// TIA Portal V19 export
DATA_BLOCK "DB_Recipes"   // DB50
{ S7_Optimized_Access := 'TRUE' }
// stored: AutoNumber false, IsOnlyStoredInLoadMemory true, MemoryReserve 100
   VAR RETAIN
      aRecipe : Array[0..256] of "stRecipe";
   END_VAR
BEGIN
   aRecipe[1].RecipeName := 'Test Flate Plate';
   aRecipe[2].RecipeName := 'Test Carbody Shell';
   aRecipe[3].RecipeName := 'RGCC5';
   aRecipe[4..23].RecipeName := '';
   aRecipe[1].RecipeCbsType := 'Flate plate';
   aRecipe[2].RecipeCbsType := 'Carbody shell';
   aRecipe[3].RecipeCbsType := 'RGC';
   aRecipe[4..5].RecipeCbsType := '';
   aRecipe[7..23].RecipeCbsType := '';
   aRecipe[1].RecipeTrajNumber := 100;
   aRecipe[2].RecipeTrajNumber := 101;
   aRecipe[3].RecipeTrajNumber := 11;
   aRecipe[4..8].RecipeTrajNumber := 0;
   aRecipe[10..23].RecipeTrajNumber := 0;
   aRecipe[1..3].RecipeRawMaterial := 1;
   aRecipe[4..8].RecipeRawMaterial := 0;
   aRecipe[10..23].RecipeRawMaterial := 0;
   aRecipe[4].RecipeLayerType[1].RecipeLayerTypeName := '';
   aRecipe[5].RecipeLayerType[1].RecipeLayerTypeName := '';
   aRecipe[6].RecipeLayerType[1].RecipeLayerTypeName := '';
   aRecipe[7].RecipeLayerType[1].RecipeLayerTypeName := '';
   aRecipe[8].RecipeLayerType[1].RecipeLayerTypeName := '';
   aRecipe[9].RecipeLayerType[1].RecipeLayerTypeName := '';
   aRecipe[10].RecipeLayerType[1].RecipeLayerTypeName := '';
   aRecipe[11].RecipeLayerType[1].RecipeLayerTypeName := '';
   aRecipe[12].RecipeLayerType[1].RecipeLayerTypeName := '';
   aRecipe[13].RecipeLayerType[1].RecipeLayerTypeName := '';
   aRecipe[14].RecipeLayerType[1].RecipeLayerTypeName := '';
   aRecipe[15].RecipeLayerType[1].RecipeLayerTypeName := '';
   aRecipe[16].RecipeLayerType[1].RecipeLayerTypeName := '';
   aRecipe[17].RecipeLayerType[1].RecipeLayerTypeName := '';
   aRecipe[18].RecipeLayerType[1].RecipeLayerTypeName := '';
   aRecipe[19].RecipeLayerType[1].RecipeLayerTypeName := '';
   aRecipe[20].RecipeLayerType[1].RecipeLayerTypeName := '';
   aRecipe[21].RecipeLayerType[1].RecipeLayerTypeName := '';
   aRecipe[22].RecipeLayerType[1].RecipeLayerTypeName := '';
   aRecipe[23].RecipeLayerType[1].RecipeLayerTypeName := '';
   aRecipe[1].RecipeLayerType[1].JobTableLeft[0].SetForceZero := 0;
   aRecipe[1].RecipeLayerType[1].JobTableLeft[1..4].SetForceZero := 100;
   aRecipe[1].RecipeLayerType[2].JobTableLeft[0].SetForceZero := 0;
   aRecipe[1].RecipeLayerType[2].JobTableLeft[1].SetForceZero := 100;
   aRecipe[1].RecipeLayerType[2].JobTableLeft[2..3].SetForceZero := 90;
   aRecipe[2].RecipeLayerType[1].JobTableLeft[0].SetForceZero := 0;
   aRecipe[2].RecipeLayerType[1].JobTableLeft[1].SetForceZero := 50;
   aRecipe[2].RecipeLayerType[2].JobTableLeft[0].SetForceZero := 0;
   aRecipe[2].RecipeLayerType[2].JobTableLeft[1].SetForceZero := 100;
   aRecipe[2].RecipeLayerType[2].JobTableLeft[2..3].SetForceZero := 80;
   aRecipe[3].RecipeLayerType[1].JobTableLeft[0].SetForceZero := 0;
   aRecipe[3].RecipeLayerType[1].JobTableLeft[1..2].SetForceZero := 80;
   aRecipe[3].RecipeLayerType[2].JobTableLeft[0].SetForceZero := 0;
   aRecipe[3].RecipeLayerType[2].JobTableLeft[1].SetForceZero := 80;
   aRecipe[4].RecipeLayerType[1].JobTableLeft[0].SetForceZero := 0;
   aRecipe[4].RecipeLayerType[2].JobTableLeft[0].SetForceZero := 0;
   aRecipe[5].RecipeLayerType[1].JobTableLeft[0].SetForceZero := 0;
   aRecipe[5].RecipeLayerType[2].JobTableLeft[0].SetForceZero := 0;
   aRecipe[6].RecipeLayerType[1].JobTableLeft[0].SetForceZero := 0;
   aRecipe[6].RecipeLayerType[1].JobTableLeft[1].SetForceZero := 20;
   aRecipe[6].RecipeLayerType[2].JobTableLeft[0].SetForceZero := 0;
   aRecipe[6].RecipeLayerType[2].JobTableLeft[1].SetForceZero := 20;
   aRecipe[7].RecipeLayerType[1].JobTableLeft[0].SetForceZero := 0;
   aRecipe[7].RecipeLayerType[2].JobTableLeft[0].SetForceZero := 0;
   aRecipe[8].RecipeLayerType[1].JobTableLeft[0].SetForceZero := 0;
   aRecipe[8].RecipeLayerType[2].JobTableLeft[0].SetForceZero := 0;
   aRecipe[9].RecipeLayerType[1].JobTableLeft[0].SetForceZero := 0;
   aRecipe[9].RecipeLayerType[2].JobTableLeft[0].SetForceZero := 0;
   aRecipe[10].RecipeLayerType[1].JobTableLeft[0].SetForceZero := 0;
   aRecipe[10].RecipeLayerType[2].JobTableLeft[0].SetForceZero := 0;
   aRecipe[11].RecipeLayerType[1].JobTableLeft[0].SetForceZero := 0;
   aRecipe[11].RecipeLayerType[2].JobTableLeft[0].SetForceZero := 0;
   aRecipe[12].RecipeLayerType[1].JobTableLeft[0].SetForceZero := 0;
   aRecipe[12].RecipeLayerType[2].JobTableLeft[0].SetForceZero := 0;
   aRecipe[13].RecipeLayerType[1].JobTableLeft[0].SetForceZero := 0;
   aRecipe[13].RecipeLayerType[2].JobTableLeft[0].SetForceZero := 0;
   aRecipe[14].RecipeLayerType[1].JobTableLeft[0].SetForceZero := 0;
   aRecipe[14].RecipeLayerType[2].JobTableLeft[0].SetForceZero := 0;
   aRecipe[15].RecipeLayerType[1].JobTableLeft[0].SetForceZero := 0;
   aRecipe[15].RecipeLayerType[2].JobTableLeft[0].SetForceZero := 0;
   aRecipe[16].RecipeLayerType[1].JobTableLeft[0].SetForceZero := 0;
   aRecipe[16].RecipeLayerType[2].JobTableLeft[0].SetForceZero := 0;
   aRecipe[17].RecipeLayerType[1].JobTableLeft[0].SetForceZero := 0;
   aRecipe[17].RecipeLayerType[2].JobTableLeft[0].SetForceZero := 0;
   aRecipe[18].RecipeLayerType[1].JobTableLeft[0].SetForceZero := 0;
   aRecipe[18].RecipeLayerType[2].JobTableLeft[0].SetForceZero := 0;
   aRecipe[19].RecipeLayerType[1].JobTableLeft[0].SetForceZero := 0;
   aRecipe[19].RecipeLayerType[2].JobTableLeft[0].SetForceZero := 0;
   aRecipe[20].RecipeLayerType[1].JobTableLeft[0].SetForceZero := 0;
   aRecipe[20].RecipeLayerType[2].JobTableLeft[0].SetForceZero := 0;
   aRecipe[21].RecipeLayerType[1].JobTableLeft[0].SetForceZero := 0;
   aRecipe[21].RecipeLayerType[2].JobTableLeft[0].SetForceZero := 0;
   aRecipe[22].RecipeLayerType[1].JobTableLeft[0].SetForceZero := 0;
   aRecipe[22].RecipeLayerType[2].JobTableLeft[0].SetForceZero := 0;
   aRecipe[23].RecipeLayerType[1].JobTableLeft[0].SetForceZero := 0;
   aRecipe[23].RecipeLayerType[2].JobTableLeft[0].SetForceZero := 0;
   aRecipe[1].RecipeLayerType[1].JobTableLeft[0].SetForceTarget := 0;
   aRecipe[1].RecipeLayerType[1].JobTableLeft[1..4].SetForceTarget := 200;
   aRecipe[1].RecipeLayerType[2].JobTableLeft[0].SetForceTarget := 0;
   aRecipe[1].RecipeLayerType[2].JobTableLeft[1].SetForceTarget := 200;
   aRecipe[1].RecipeLayerType[2].JobTableLeft[2].SetForceTarget := 150;
   aRecipe[1].RecipeLayerType[2].JobTableLeft[3].SetForceTarget := 180;
   aRecipe[2].RecipeLayerType[1].JobTableLeft[0].SetForceTarget := 0;
   aRecipe[2].RecipeLayerType[1].JobTableLeft[1].SetForceTarget := 80;
   aRecipe[2].RecipeLayerType[2].JobTableLeft[0].SetForceTarget := 0;
   aRecipe[2].RecipeLayerType[2].JobTableLeft[1].SetForceTarget := 200;
   aRecipe[2].RecipeLayerType[2].JobTableLeft[3].SetForceTarget := 150;
   aRecipe[3].RecipeLayerType[1].JobTableLeft[0].SetForceTarget := 0;
   aRecipe[3].RecipeLayerType[1].JobTableLeft[1..2].SetForceTarget := 120;
   aRecipe[3].RecipeLayerType[2].JobTableLeft[0].SetForceTarget := 0;
   aRecipe[3].RecipeLayerType[2].JobTableLeft[1].SetForceTarget := 120;
   aRecipe[4].RecipeLayerType[1].JobTableLeft[0].SetForceTarget := 0;
   aRecipe[4].RecipeLayerType[2].JobTableLeft[0].SetForceTarget := 0;
   aRecipe[5].RecipeLayerType[1].JobTableLeft[0].SetForceTarget := 0;
   aRecipe[5].RecipeLayerType[2].JobTableLeft[0].SetForceTarget := 0;
   aRecipe[6].RecipeLayerType[1].JobTableLeft[0].SetForceTarget := 0;
   aRecipe[6].RecipeLayerType[1].JobTableLeft[1].SetForceTarget := 120;
   aRecipe[6].RecipeLayerType[2].JobTableLeft[0].SetForceTarget := 0;
   aRecipe[6].RecipeLayerType[2].JobTableLeft[1].SetForceTarget := 120;
   aRecipe[7].RecipeLayerType[1].JobTableLeft[0].SetForceTarget := 0;
   aRecipe[7].RecipeLayerType[2].JobTableLeft[0].SetForceTarget := 0;
   aRecipe[8].RecipeLayerType[1].JobTableLeft[0].SetForceTarget := 0;
   aRecipe[8].RecipeLayerType[2].JobTableLeft[0].SetForceTarget := 0;
   aRecipe[9].RecipeLayerType[1].JobTableLeft[0].SetForceTarget := 0;
   aRecipe[9].RecipeLayerType[2].JobTableLeft[0].SetForceTarget := 0;
   aRecipe[10].RecipeLayerType[1].JobTableLeft[0].SetForceTarget := 0;
   aRecipe[10].RecipeLayerType[2].JobTableLeft[0].SetForceTarget := 0;
   aRecipe[11].RecipeLayerType[1].JobTableLeft[0].SetForceTarget := 0;
   aRecipe[11].RecipeLayerType[2].JobTableLeft[0].SetForceTarget := 0;
   aRecipe[12].RecipeLayerType[1].JobTableLeft[0].SetForceTarget := 0;
   aRecipe[12].RecipeLayerType[2].JobTableLeft[0].SetForceTarget := 0;
   aRecipe[13].RecipeLayerType[1].JobTableLeft[0].SetForceTarget := 0;
   aRecipe[13].RecipeLayerType[2].JobTableLeft[0].SetForceTarget := 0;
   aRecipe[14].RecipeLayerType[1].JobTableLeft[0].SetForceTarget := 0;
   aRecipe[14].RecipeLayerType[2].JobTableLeft[0].SetForceTarget := 0;
   aRecipe[15].RecipeLayerType[1].JobTableLeft[0].SetForceTarget := 0;
   aRecipe[15].RecipeLayerType[2].JobTableLeft[0].SetForceTarget := 0;
   aRecipe[16].RecipeLayerType[1].JobTableLeft[0].SetForceTarget := 0;
   aRecipe[16].RecipeLayerType[2].JobTableLeft[0].SetForceTarget := 0;
   aRecipe[17].RecipeLayerType[1].JobTableLeft[0].SetForceTarget := 0;
   aRecipe[17].RecipeLayerType[2].JobTableLeft[0].SetForceTarget := 0;
   aRecipe[18].RecipeLayerType[1].JobTableLeft[0].SetForceTarget := 0;
   aRecipe[18].RecipeLayerType[2].JobTableLeft[0].SetForceTarget := 0;
   aRecipe[19].RecipeLayerType[1].JobTableLeft[0].SetForceTarget := 0;
   aRecipe[19].RecipeLayerType[2].JobTableLeft[0].SetForceTarget := 0;
   aRecipe[20].RecipeLayerType[1].JobTableLeft[0].SetForceTarget := 0;
   aRecipe[20].RecipeLayerType[2].JobTableLeft[0].SetForceTarget := 0;
   aRecipe[21].RecipeLayerType[1].JobTableLeft[0].SetForceTarget := 0;
   aRecipe[21].RecipeLayerType[2].JobTableLeft[0].SetForceTarget := 0;
   aRecipe[22].RecipeLayerType[1].JobTableLeft[0].SetForceTarget := 0;
   aRecipe[22].RecipeLayerType[2].JobTableLeft[0].SetForceTarget := 0;
   aRecipe[23].RecipeLayerType[1].JobTableLeft[0].SetForceTarget := 0;
   aRecipe[23].RecipeLayerType[2].JobTableLeft[0].SetForceTarget := 0;
   aRecipe[1].RecipeLayerType[1].JobTableLeft[0].SetTimeRamp := 0;
   aRecipe[1].RecipeLayerType[2].JobTableLeft[0].SetTimeRamp := 0;
   aRecipe[2].RecipeLayerType[1].JobTableLeft[0].SetTimeRamp := 0;
   aRecipe[2].RecipeLayerType[2].JobTableLeft[0].SetTimeRamp := 0;
   aRecipe[3].RecipeLayerType[1].JobTableLeft[0].SetTimeRamp := 0;
   aRecipe[3].RecipeLayerType[2].JobTableLeft[0].SetTimeRamp := 0;
   aRecipe[4].RecipeLayerType[1].JobTableLeft[0].SetTimeRamp := 0;
   aRecipe[4].RecipeLayerType[2].JobTableLeft[0].SetTimeRamp := 0;
   aRecipe[5].RecipeLayerType[1].JobTableLeft[0].SetTimeRamp := 0;
   aRecipe[5].RecipeLayerType[2].JobTableLeft[0].SetTimeRamp := 0;
   aRecipe[6].RecipeLayerType[1].JobTableLeft[0].SetTimeRamp := 0;
   aRecipe[6].RecipeLayerType[2].JobTableLeft[0].SetTimeRamp := 0;
   aRecipe[7].RecipeLayerType[1].JobTableLeft[0].SetTimeRamp := 0;
   aRecipe[7].RecipeLayerType[2].JobTableLeft[0].SetTimeRamp := 0;
   aRecipe[8].RecipeLayerType[1].JobTableLeft[0].SetTimeRamp := 0;
   aRecipe[8].RecipeLayerType[2].JobTableLeft[0].SetTimeRamp := 0;
   aRecipe[9].RecipeLayerType[1].JobTableLeft[0].SetTimeRamp := 0;
   aRecipe[9].RecipeLayerType[2].JobTableLeft[0].SetTimeRamp := 0;
   aRecipe[10].RecipeLayerType[1].JobTableLeft[0].SetTimeRamp := 0;
   aRecipe[10].RecipeLayerType[2].JobTableLeft[0].SetTimeRamp := 0;
   aRecipe[11].RecipeLayerType[1].JobTableLeft[0].SetTimeRamp := 0;
   aRecipe[11].RecipeLayerType[2].JobTableLeft[0].SetTimeRamp := 0;
   aRecipe[12].RecipeLayerType[1].JobTableLeft[0].SetTimeRamp := 0;
   aRecipe[12].RecipeLayerType[2].JobTableLeft[0].SetTimeRamp := 0;
   aRecipe[13].RecipeLayerType[1].JobTableLeft[0].SetTimeRamp := 0;
   aRecipe[13].RecipeLayerType[2].JobTableLeft[0].SetTimeRamp := 0;
   aRecipe[14].RecipeLayerType[1].JobTableLeft[0].SetTimeRamp := 0;
   aRecipe[14].RecipeLayerType[2].JobTableLeft[0].SetTimeRamp := 0;
   aRecipe[15].RecipeLayerType[1].JobTableLeft[0].SetTimeRamp := 0;
   aRecipe[15].RecipeLayerType[2].JobTableLeft[0].SetTimeRamp := 0;
   aRecipe[16].RecipeLayerType[1].JobTableLeft[0].SetTimeRamp := 0;
   aRecipe[16].RecipeLayerType[2].JobTableLeft[0].SetTimeRamp := 0;
   aRecipe[17].RecipeLayerType[1].JobTableLeft[0].SetTimeRamp := 0;
   aRecipe[17].RecipeLayerType[2].JobTableLeft[0].SetTimeRamp := 0;
   aRecipe[18].RecipeLayerType[1].JobTableLeft[0].SetTimeRamp := 0;
   aRecipe[18].RecipeLayerType[2].JobTableLeft[0].SetTimeRamp := 0;
   aRecipe[19].RecipeLayerType[1].JobTableLeft[0].SetTimeRamp := 0;
   aRecipe[19].RecipeLayerType[2].JobTableLeft[0].SetTimeRamp := 0;
   aRecipe[20].RecipeLayerType[1].JobTableLeft[0].SetTimeRamp := 0;
   aRecipe[20].RecipeLayerType[2].JobTableLeft[0].SetTimeRamp := 0;
   aRecipe[21].RecipeLayerType[1].JobTableLeft[0].SetTimeRamp := 0;
   aRecipe[21].RecipeLayerType[2].JobTableLeft[0].SetTimeRamp := 0;
   aRecipe[22].RecipeLayerType[1].JobTableLeft[0].SetTimeRamp := 0;
   aRecipe[22].RecipeLayerType[2].JobTableLeft[0].SetTimeRamp := 0;
   aRecipe[23].RecipeLayerType[1].JobTableLeft[0].SetTimeRamp := 0;
   aRecipe[23].RecipeLayerType[2].JobTableLeft[0].SetTimeRamp := 0;
   aRecipe[1].RecipeLayerType[1].JobTableLeft[0].SetSpeed := 0;
   aRecipe[1].RecipeLayerType[1].JobTableLeft[3..4].SetSpeed := 5000;
   aRecipe[1].RecipeLayerType[2].JobTableLeft[0].SetSpeed := 0;
   aRecipe[2].RecipeLayerType[1].JobTableLeft[0].SetSpeed := 0;
   aRecipe[2].RecipeLayerType[2].JobTableLeft[0].SetSpeed := 0;
   aRecipe[3].RecipeLayerType[1].JobTableLeft[0].SetSpeed := 0;
   aRecipe[3].RecipeLayerType[2].JobTableLeft[0].SetSpeed := 0;
   aRecipe[4].RecipeLayerType[1].JobTableLeft[0].SetSpeed := 0;
   aRecipe[4].RecipeLayerType[2].JobTableLeft[0].SetSpeed := 0;
   aRecipe[5].RecipeLayerType[1].JobTableLeft[0].SetSpeed := 0;
   aRecipe[5].RecipeLayerType[2].JobTableLeft[0].SetSpeed := 0;
   aRecipe[6].RecipeLayerType[1].JobTableLeft[0].SetSpeed := 0;
   aRecipe[6].RecipeLayerType[2].JobTableLeft[0].SetSpeed := 0;
   aRecipe[7].RecipeLayerType[1].JobTableLeft[0].SetSpeed := 0;
   aRecipe[7].RecipeLayerType[2].JobTableLeft[0].SetSpeed := 0;
   aRecipe[8].RecipeLayerType[1].JobTableLeft[0].SetSpeed := 0;
   aRecipe[8].RecipeLayerType[2].JobTableLeft[0].SetSpeed := 0;
   aRecipe[9].RecipeLayerType[1].JobTableLeft[0].SetSpeed := 0;
   aRecipe[9].RecipeLayerType[2].JobTableLeft[0].SetSpeed := 0;
   aRecipe[10].RecipeLayerType[1].JobTableLeft[0].SetSpeed := 0;
   aRecipe[10].RecipeLayerType[2].JobTableLeft[0].SetSpeed := 0;
   aRecipe[11].RecipeLayerType[1].JobTableLeft[0].SetSpeed := 0;
   aRecipe[11].RecipeLayerType[2].JobTableLeft[0].SetSpeed := 0;
   aRecipe[12].RecipeLayerType[1].JobTableLeft[0].SetSpeed := 0;
   aRecipe[12].RecipeLayerType[2].JobTableLeft[0].SetSpeed := 0;
   aRecipe[13].RecipeLayerType[1].JobTableLeft[0].SetSpeed := 0;
   aRecipe[13].RecipeLayerType[2].JobTableLeft[0].SetSpeed := 0;
   aRecipe[14].RecipeLayerType[1].JobTableLeft[0].SetSpeed := 0;
   aRecipe[14].RecipeLayerType[2].JobTableLeft[0].SetSpeed := 0;
   aRecipe[15].RecipeLayerType[1].JobTableLeft[0].SetSpeed := 0;
   aRecipe[15].RecipeLayerType[2].JobTableLeft[0].SetSpeed := 0;
   aRecipe[16].RecipeLayerType[1].JobTableLeft[0].SetSpeed := 0;
   aRecipe[16].RecipeLayerType[2].JobTableLeft[0].SetSpeed := 0;
   aRecipe[17].RecipeLayerType[1].JobTableLeft[0].SetSpeed := 0;
   aRecipe[17].RecipeLayerType[2].JobTableLeft[0].SetSpeed := 0;
   aRecipe[18].RecipeLayerType[1].JobTableLeft[0].SetSpeed := 0;
   aRecipe[18].RecipeLayerType[2].JobTableLeft[0].SetSpeed := 0;
   aRecipe[19].RecipeLayerType[1].JobTableLeft[0].SetSpeed := 0;
   aRecipe[19].RecipeLayerType[2].JobTableLeft[0].SetSpeed := 0;
   aRecipe[20].RecipeLayerType[1].JobTableLeft[0].SetSpeed := 0;
   aRecipe[20].RecipeLayerType[2].JobTableLeft[0].SetSpeed := 0;
   aRecipe[21].RecipeLayerType[1].JobTableLeft[0].SetSpeed := 0;
   aRecipe[21].RecipeLayerType[2].JobTableLeft[0].SetSpeed := 0;
   aRecipe[22].RecipeLayerType[1].JobTableLeft[0].SetSpeed := 0;
   aRecipe[22].RecipeLayerType[2].JobTableLeft[0].SetSpeed := 0;
   aRecipe[23].RecipeLayerType[1].JobTableLeft[0].SetSpeed := 0;
   aRecipe[23].RecipeLayerType[2].JobTableLeft[0].SetSpeed := 0;
   aRecipe[1].RecipeLayerType[1].JobTableLeft[0].SetRobotSpeed := 0;
   aRecipe[1].RecipeLayerType[1].JobTableLeft[1].SetRobotSpeed := 300;
   aRecipe[1].RecipeLayerType[1].JobTableLeft[2].SetRobotSpeed := 500;
   aRecipe[1].RecipeLayerType[1].JobTableLeft[3..4].SetRobotSpeed := 300;
   aRecipe[1].RecipeLayerType[2].JobTableLeft[0].SetRobotSpeed := 0;
   aRecipe[1].RecipeLayerType[2].JobTableLeft[1..3].SetRobotSpeed := 300;
   aRecipe[2].RecipeLayerType[1].JobTableLeft[0].SetRobotSpeed := 0;
   aRecipe[2].RecipeLayerType[1].JobTableLeft[1].SetRobotSpeed := 300;
   aRecipe[2].RecipeLayerType[2].JobTableLeft[0].SetRobotSpeed := 0;
   aRecipe[2].RecipeLayerType[2].JobTableLeft[1..2].SetRobotSpeed := 300;
   aRecipe[2].RecipeLayerType[2].JobTableLeft[3].SetRobotSpeed := 250;
   aRecipe[3].RecipeLayerType[1].JobTableLeft[0].SetRobotSpeed := 0;
   aRecipe[3].RecipeLayerType[1].JobTableLeft[1].SetRobotSpeed := 200;
   aRecipe[3].RecipeLayerType[1].JobTableLeft[2].SetRobotSpeed := 300;
   aRecipe[3].RecipeLayerType[2].JobTableLeft[0].SetRobotSpeed := 0;
   aRecipe[3].RecipeLayerType[2].JobTableLeft[1].SetRobotSpeed := 300;
   aRecipe[4].RecipeLayerType[1].JobTableLeft[0].SetRobotSpeed := 0;
   aRecipe[4].RecipeLayerType[2].JobTableLeft[0].SetRobotSpeed := 0;
   aRecipe[5].RecipeLayerType[1].JobTableLeft[0].SetRobotSpeed := 0;
   aRecipe[5].RecipeLayerType[2].JobTableLeft[0].SetRobotSpeed := 0;
   aRecipe[6].RecipeLayerType[1].JobTableLeft[0].SetRobotSpeed := 0;
   aRecipe[6].RecipeLayerType[2].JobTableLeft[0].SetRobotSpeed := 0;
   aRecipe[7].RecipeLayerType[1].JobTableLeft[0].SetRobotSpeed := 0;
   aRecipe[7].RecipeLayerType[2].JobTableLeft[0].SetRobotSpeed := 0;
   aRecipe[8].RecipeLayerType[1].JobTableLeft[0].SetRobotSpeed := 0;
   aRecipe[8].RecipeLayerType[2].JobTableLeft[0].SetRobotSpeed := 0;
   aRecipe[9].RecipeLayerType[1].JobTableLeft[0].SetRobotSpeed := 0;
   aRecipe[9].RecipeLayerType[2].JobTableLeft[0].SetRobotSpeed := 0;
   aRecipe[10].RecipeLayerType[1].JobTableLeft[0].SetRobotSpeed := 0;
   aRecipe[10].RecipeLayerType[2].JobTableLeft[0].SetRobotSpeed := 0;
   aRecipe[11].RecipeLayerType[1].JobTableLeft[0].SetRobotSpeed := 0;
   aRecipe[11].RecipeLayerType[2].JobTableLeft[0].SetRobotSpeed := 0;
   aRecipe[12].RecipeLayerType[1].JobTableLeft[0].SetRobotSpeed := 0;
   aRecipe[12].RecipeLayerType[2].JobTableLeft[0].SetRobotSpeed := 0;
   aRecipe[13].RecipeLayerType[1].JobTableLeft[0].SetRobotSpeed := 0;
   aRecipe[13].RecipeLayerType[2].JobTableLeft[0].SetRobotSpeed := 0;
   aRecipe[14].RecipeLayerType[1].JobTableLeft[0].SetRobotSpeed := 0;
   aRecipe[14].RecipeLayerType[2].JobTableLeft[0].SetRobotSpeed := 0;
   aRecipe[15].RecipeLayerType[1].JobTableLeft[0].SetRobotSpeed := 0;
   aRecipe[15].RecipeLayerType[2].JobTableLeft[0].SetRobotSpeed := 0;
   aRecipe[16].RecipeLayerType[1].JobTableLeft[0].SetRobotSpeed := 0;
   aRecipe[16].RecipeLayerType[2].JobTableLeft[0].SetRobotSpeed := 0;
   aRecipe[17].RecipeLayerType[1].JobTableLeft[0].SetRobotSpeed := 0;
   aRecipe[17].RecipeLayerType[2].JobTableLeft[0].SetRobotSpeed := 0;
   aRecipe[18].RecipeLayerType[1].JobTableLeft[0].SetRobotSpeed := 0;
   aRecipe[18].RecipeLayerType[2].JobTableLeft[0].SetRobotSpeed := 0;
   aRecipe[19].RecipeLayerType[1].JobTableLeft[0].SetRobotSpeed := 0;
   aRecipe[19].RecipeLayerType[2].JobTableLeft[0].SetRobotSpeed := 0;
   aRecipe[20].RecipeLayerType[1].JobTableLeft[0].SetRobotSpeed := 0;
   aRecipe[20].RecipeLayerType[2].JobTableLeft[0].SetRobotSpeed := 0;
   aRecipe[21].RecipeLayerType[1].JobTableLeft[0].SetRobotSpeed := 0;
   aRecipe[21].RecipeLayerType[2].JobTableLeft[0].SetRobotSpeed := 0;
   aRecipe[22].RecipeLayerType[1].JobTableLeft[0].SetRobotSpeed := 0;
   aRecipe[22].RecipeLayerType[2].JobTableLeft[0].SetRobotSpeed := 0;
   aRecipe[23].RecipeLayerType[1].JobTableLeft[0].SetRobotSpeed := 0;
   aRecipe[23].RecipeLayerType[2].JobTableLeft[0].SetRobotSpeed := 0;
   aRecipe[1].RecipeLayerType[1].JobTableLeft[0].WornPaperDistance := 0;
   aRecipe[1].RecipeLayerType[1].JobTableLeft[1..4].WornPaperDistance := 900;
   aRecipe[1].RecipeLayerType[2].JobTableLeft[0].WornPaperDistance := 0;
   aRecipe[1].RecipeLayerType[2].JobTableLeft[1..3].WornPaperDistance := 900;
   aRecipe[2].RecipeLayerType[1].JobTableLeft[0].WornPaperDistance := 0;
   aRecipe[2].RecipeLayerType[1].JobTableLeft[1].WornPaperDistance := 8;
   aRecipe[2].RecipeLayerType[1].JobTableLeft[2..3].WornPaperDistance := 999;
   aRecipe[2].RecipeLayerType[2].JobTableLeft[0].WornPaperDistance := 0;
   aRecipe[2].RecipeLayerType[2].JobTableLeft[1..2].WornPaperDistance := 30;
   aRecipe[2].RecipeLayerType[2].JobTableLeft[3].WornPaperDistance := 999;
   aRecipe[3].RecipeLayerType[1].JobTableLeft[0].WornPaperDistance := 0;
   aRecipe[3].RecipeLayerType[1].JobTableLeft[1..2].WornPaperDistance := 30;
   aRecipe[3].RecipeLayerType[2].JobTableLeft[0].WornPaperDistance := 0;
   aRecipe[3].RecipeLayerType[2].JobTableLeft[1].WornPaperDistance := 30;
   aRecipe[4].RecipeLayerType[1].JobTableLeft[0].WornPaperDistance := 0;
   aRecipe[4].RecipeLayerType[2].JobTableLeft[0].WornPaperDistance := 0;
   aRecipe[5].RecipeLayerType[1].JobTableLeft[0].WornPaperDistance := 0;
   aRecipe[5].RecipeLayerType[2].JobTableLeft[0].WornPaperDistance := 0;
   aRecipe[6].RecipeLayerType[1].JobTableLeft[0].WornPaperDistance := 0;
   aRecipe[6].RecipeLayerType[2].JobTableLeft[0].WornPaperDistance := 0;
   aRecipe[7].RecipeLayerType[1].JobTableLeft[0].WornPaperDistance := 0;
   aRecipe[7].RecipeLayerType[2].JobTableLeft[0].WornPaperDistance := 0;
   aRecipe[8].RecipeLayerType[1].JobTableLeft[0].WornPaperDistance := 0;
   aRecipe[8].RecipeLayerType[2].JobTableLeft[0].WornPaperDistance := 0;
   aRecipe[9].RecipeLayerType[1].JobTableLeft[0].WornPaperDistance := 0;
   aRecipe[9].RecipeLayerType[2].JobTableLeft[0].WornPaperDistance := 0;
   aRecipe[10].RecipeLayerType[1].JobTableLeft[0].WornPaperDistance := 0;
   aRecipe[10].RecipeLayerType[2].JobTableLeft[0].WornPaperDistance := 0;
   aRecipe[11].RecipeLayerType[1].JobTableLeft[0].WornPaperDistance := 0;
   aRecipe[11].RecipeLayerType[2].JobTableLeft[0].WornPaperDistance := 0;
   aRecipe[12].RecipeLayerType[1].JobTableLeft[0].WornPaperDistance := 0;
   aRecipe[12].RecipeLayerType[2].JobTableLeft[0].WornPaperDistance := 0;
   aRecipe[13].RecipeLayerType[1].JobTableLeft[0].WornPaperDistance := 0;
   aRecipe[13].RecipeLayerType[2].JobTableLeft[0].WornPaperDistance := 0;
   aRecipe[14].RecipeLayerType[1].JobTableLeft[0].WornPaperDistance := 0;
   aRecipe[14].RecipeLayerType[2].JobTableLeft[0].WornPaperDistance := 0;
   aRecipe[15].RecipeLayerType[1].JobTableLeft[0].WornPaperDistance := 0;
   aRecipe[15].RecipeLayerType[2].JobTableLeft[0].WornPaperDistance := 0;
   aRecipe[16].RecipeLayerType[1].JobTableLeft[0].WornPaperDistance := 0;
   aRecipe[16].RecipeLayerType[2].JobTableLeft[0].WornPaperDistance := 0;
   aRecipe[17].RecipeLayerType[1].JobTableLeft[0].WornPaperDistance := 0;
   aRecipe[17].RecipeLayerType[2].JobTableLeft[0].WornPaperDistance := 0;
   aRecipe[18].RecipeLayerType[1].JobTableLeft[0].WornPaperDistance := 0;
   aRecipe[18].RecipeLayerType[2].JobTableLeft[0].WornPaperDistance := 0;
   aRecipe[19].RecipeLayerType[1].JobTableLeft[0].WornPaperDistance := 0;
   aRecipe[19].RecipeLayerType[2].JobTableLeft[0].WornPaperDistance := 0;
   aRecipe[20].RecipeLayerType[1].JobTableLeft[0].WornPaperDistance := 0;
   aRecipe[20].RecipeLayerType[2].JobTableLeft[0].WornPaperDistance := 0;
   aRecipe[21].RecipeLayerType[1].JobTableLeft[0].WornPaperDistance := 0;
   aRecipe[21].RecipeLayerType[2].JobTableLeft[0].WornPaperDistance := 0;
   aRecipe[22].RecipeLayerType[1].JobTableLeft[0].WornPaperDistance := 0;
   aRecipe[22].RecipeLayerType[2].JobTableLeft[0].WornPaperDistance := 0;
   aRecipe[23].RecipeLayerType[1].JobTableLeft[0].WornPaperDistance := 0;
   aRecipe[23].RecipeLayerType[2].JobTableLeft[0].WornPaperDistance := 0;
   aRecipe[1].RecipeLayerType[1].JobTableLeft[0].Gimball := 0;
   aRecipe[1].RecipeLayerType[2].JobTableLeft[0].Gimball := 0;
   aRecipe[2].RecipeLayerType[1].JobTableLeft[0].Gimball := 0;
   aRecipe[2].RecipeLayerType[2].JobTableLeft[0].Gimball := 0;
   aRecipe[3].RecipeLayerType[1].JobTableLeft[0].Gimball := 0;
   aRecipe[3].RecipeLayerType[2].JobTableLeft[0].Gimball := 0;
   aRecipe[3].RecipeLayerType[2].JobTableLeft[1].Gimball := 1;
   aRecipe[4].RecipeLayerType[1].JobTableLeft[0].Gimball := 0;
   aRecipe[4].RecipeLayerType[2].JobTableLeft[0].Gimball := 0;
   aRecipe[5].RecipeLayerType[1].JobTableLeft[0].Gimball := 0;
   aRecipe[5].RecipeLayerType[2].JobTableLeft[0].Gimball := 0;
   aRecipe[6].RecipeLayerType[1].JobTableLeft[0].Gimball := 0;
   aRecipe[6].RecipeLayerType[2].JobTableLeft[0].Gimball := 0;
   aRecipe[7].RecipeLayerType[1].JobTableLeft[0].Gimball := 0;
   aRecipe[7].RecipeLayerType[2].JobTableLeft[0].Gimball := 0;
   aRecipe[8].RecipeLayerType[1].JobTableLeft[0].Gimball := 0;
   aRecipe[8].RecipeLayerType[2].JobTableLeft[0].Gimball := 0;
   aRecipe[9].RecipeLayerType[1].JobTableLeft[0].Gimball := 0;
   aRecipe[9].RecipeLayerType[2].JobTableLeft[0].Gimball := 0;
   aRecipe[10].RecipeLayerType[1].JobTableLeft[0].Gimball := 0;
   aRecipe[10].RecipeLayerType[2].JobTableLeft[0].Gimball := 0;
   aRecipe[11].RecipeLayerType[1].JobTableLeft[0].Gimball := 0;
   aRecipe[11].RecipeLayerType[2].JobTableLeft[0].Gimball := 0;
   aRecipe[12].RecipeLayerType[1].JobTableLeft[0].Gimball := 0;
   aRecipe[12].RecipeLayerType[2].JobTableLeft[0].Gimball := 0;
   aRecipe[13].RecipeLayerType[1].JobTableLeft[0].Gimball := 0;
   aRecipe[13].RecipeLayerType[2].JobTableLeft[0].Gimball := 0;
   aRecipe[14].RecipeLayerType[1].JobTableLeft[0].Gimball := 0;
   aRecipe[14].RecipeLayerType[2].JobTableLeft[0].Gimball := 0;
   aRecipe[15].RecipeLayerType[1].JobTableLeft[0].Gimball := 0;
   aRecipe[15].RecipeLayerType[2].JobTableLeft[0].Gimball := 0;
   aRecipe[16].RecipeLayerType[1].JobTableLeft[0].Gimball := 0;
   aRecipe[16].RecipeLayerType[2].JobTableLeft[0].Gimball := 0;
   aRecipe[17].RecipeLayerType[1].JobTableLeft[0].Gimball := 0;
   aRecipe[17].RecipeLayerType[1].JobTableLeft[1].Gimball := 1;
   aRecipe[17].RecipeLayerType[2].JobTableLeft[0].Gimball := 0;
   aRecipe[18].RecipeLayerType[1].JobTableLeft[0].Gimball := 0;
   aRecipe[18].RecipeLayerType[2].JobTableLeft[0].Gimball := 0;
   aRecipe[19].RecipeLayerType[1].JobTableLeft[0].Gimball := 0;
   aRecipe[19].RecipeLayerType[2].JobTableLeft[0].Gimball := 0;
   aRecipe[20].RecipeLayerType[1].JobTableLeft[0].Gimball := 0;
   aRecipe[20].RecipeLayerType[2].JobTableLeft[0].Gimball := 0;
   aRecipe[21].RecipeLayerType[1].JobTableLeft[0].Gimball := 0;
   aRecipe[21].RecipeLayerType[2].JobTableLeft[0].Gimball := 0;
   aRecipe[22].RecipeLayerType[1].JobTableLeft[0].Gimball := 0;
   aRecipe[22].RecipeLayerType[2].JobTableLeft[0].Gimball := 0;
   aRecipe[23].RecipeLayerType[1].JobTableLeft[0].Gimball := 0;
   aRecipe[23].RecipeLayerType[2].JobTableLeft[0].Gimball := 0;
   aRecipe[1].RecipeLayerType[1].JobTableLeft[1..4].UnlockEccentric1 := TRUE;
   aRecipe[1].RecipeLayerType[2].JobTableLeft[3].UnlockEccentric1 := TRUE;
   aRecipe[1].RecipeLayerType[1].JobTableLeft[1..4].UnlockEccentric2 := TRUE;
   aRecipe[1].RecipeLayerType[2].JobTableLeft[3].UnlockEccentric2 := TRUE;
   aRecipe[1].RecipeLayerType[1].JobTableLeft[1..4].UnlockEccentric3 := TRUE;
   aRecipe[1].RecipeLayerType[2].JobTableLeft[3].UnlockEccentric3 := TRUE;
   aRecipe[1].RecipeLayerType[1].JobTableRight[0].SetForceZero := 0;
   aRecipe[1].RecipeLayerType[1].JobTableRight[1].SetForceZero := 21;
   aRecipe[1].RecipeLayerType[1].JobTableRight[2].SetForceZero := 22;
   aRecipe[1].RecipeLayerType[2].JobTableRight[0].SetForceZero := 0;
   aRecipe[2].RecipeLayerType[1].JobTableRight[0].SetForceZero := 0;
   aRecipe[2].RecipeLayerType[1].JobTableRight[1].SetForceZero := 50;
   aRecipe[2].RecipeLayerType[1].JobTableRight[2].SetForceZero := 80;
   aRecipe[2].RecipeLayerType[1].JobTableRight[3].SetForceZero := 50;
   aRecipe[2].RecipeLayerType[2].JobTableRight[0].SetForceZero := 0;
   aRecipe[2].RecipeLayerType[2].JobTableRight[1].SetForceZero := 100;
   aRecipe[2].RecipeLayerType[2].JobTableRight[2].SetForceZero := 80;
   aRecipe[3].RecipeLayerType[1].JobTableRight[0].SetForceZero := 0;
   aRecipe[3].RecipeLayerType[1].JobTableRight[1..2].SetForceZero := 80;
   aRecipe[3].RecipeLayerType[2].JobTableRight[0].SetForceZero := 0;
   aRecipe[3].RecipeLayerType[2].JobTableRight[1].SetForceZero := 80;
   aRecipe[4].RecipeLayerType[1].JobTableRight[0].SetForceZero := 0;
   aRecipe[4].RecipeLayerType[2].JobTableRight[0].SetForceZero := 0;
   aRecipe[5].RecipeLayerType[1].JobTableRight[0].SetForceZero := 0;
   aRecipe[5].RecipeLayerType[2].JobTableRight[0].SetForceZero := 0;
   aRecipe[6].RecipeLayerType[1].JobTableRight[0].SetForceZero := 0;
   aRecipe[6].RecipeLayerType[1].JobTableRight[1].SetForceZero := 20;
   aRecipe[6].RecipeLayerType[2].JobTableRight[0].SetForceZero := 0;
   aRecipe[6].RecipeLayerType[2].JobTableRight[1].SetForceZero := 20;
   aRecipe[7].RecipeLayerType[1].JobTableRight[0].SetForceZero := 0;
   aRecipe[7].RecipeLayerType[2].JobTableRight[0].SetForceZero := 0;
   aRecipe[8].RecipeLayerType[1].JobTableRight[0].SetForceZero := 0;
   aRecipe[8].RecipeLayerType[2].JobTableRight[0].SetForceZero := 0;
   aRecipe[9].RecipeLayerType[1].JobTableRight[0].SetForceZero := 0;
   aRecipe[9].RecipeLayerType[2].JobTableRight[0].SetForceZero := 0;
   aRecipe[10].RecipeLayerType[1].JobTableRight[0].SetForceZero := 0;
   aRecipe[10].RecipeLayerType[2].JobTableRight[0].SetForceZero := 0;
   aRecipe[11].RecipeLayerType[1].JobTableRight[0].SetForceZero := 0;
   aRecipe[11].RecipeLayerType[2].JobTableRight[0].SetForceZero := 0;
   aRecipe[12].RecipeLayerType[1].JobTableRight[0].SetForceZero := 0;
   aRecipe[12].RecipeLayerType[2].JobTableRight[0].SetForceZero := 0;
   aRecipe[13].RecipeLayerType[1].JobTableRight[0].SetForceZero := 0;
   aRecipe[13].RecipeLayerType[2].JobTableRight[0].SetForceZero := 0;
   aRecipe[14].RecipeLayerType[1].JobTableRight[0].SetForceZero := 0;
   aRecipe[14].RecipeLayerType[2].JobTableRight[0].SetForceZero := 0;
   aRecipe[15].RecipeLayerType[1].JobTableRight[0].SetForceZero := 0;
   aRecipe[15].RecipeLayerType[2].JobTableRight[0].SetForceZero := 0;
   aRecipe[16].RecipeLayerType[1].JobTableRight[0].SetForceZero := 0;
   aRecipe[16].RecipeLayerType[2].JobTableRight[0].SetForceZero := 0;
   aRecipe[17].RecipeLayerType[1].JobTableRight[0].SetForceZero := 0;
   aRecipe[17].RecipeLayerType[1].JobTableRight[1].SetForceZero := 20;
   aRecipe[17].RecipeLayerType[2].JobTableRight[0].SetForceZero := 0;
   aRecipe[18].RecipeLayerType[1].JobTableRight[0].SetForceZero := 0;
   aRecipe[18].RecipeLayerType[2].JobTableRight[0].SetForceZero := 0;
   aRecipe[19].RecipeLayerType[1].JobTableRight[0].SetForceZero := 0;
   aRecipe[19].RecipeLayerType[2].JobTableRight[0].SetForceZero := 0;
   aRecipe[20].RecipeLayerType[1].JobTableRight[0].SetForceZero := 0;
   aRecipe[20].RecipeLayerType[2].JobTableRight[0].SetForceZero := 0;
   aRecipe[21].RecipeLayerType[1].JobTableRight[0].SetForceZero := 0;
   aRecipe[21].RecipeLayerType[2].JobTableRight[0].SetForceZero := 0;
   aRecipe[22].RecipeLayerType[1].JobTableRight[0].SetForceZero := 0;
   aRecipe[22].RecipeLayerType[2].JobTableRight[0].SetForceZero := 0;
   aRecipe[23].RecipeLayerType[1].JobTableRight[0].SetForceZero := 0;
   aRecipe[23].RecipeLayerType[2].JobTableRight[0].SetForceZero := 0;
   aRecipe[1].RecipeLayerType[1].JobTableRight[0].SetForceTarget := 0;
   aRecipe[1].RecipeLayerType[2].JobTableRight[0].SetForceTarget := 0;
   aRecipe[2].RecipeLayerType[1].JobTableRight[0].SetForceTarget := 0;
   aRecipe[2].RecipeLayerType[1].JobTableRight[1].SetForceTarget := 80;
   aRecipe[2].RecipeLayerType[1].JobTableRight[3].SetForceTarget := 100;
   aRecipe[2].RecipeLayerType[2].JobTableRight[0].SetForceTarget := 0;
   aRecipe[2].RecipeLayerType[2].JobTableRight[1].SetForceTarget := 200;
   aRecipe[3].RecipeLayerType[1].JobTableRight[0].SetForceTarget := 0;
   aRecipe[3].RecipeLayerType[1].JobTableRight[1].SetForceTarget := 120;
   aRecipe[3].RecipeLayerType[2].JobTableRight[0].SetForceTarget := 0;
   aRecipe[3].RecipeLayerType[2].JobTableRight[1].SetForceTarget := 120;
   aRecipe[4].RecipeLayerType[1].JobTableRight[0].SetForceTarget := 0;
   aRecipe[4].RecipeLayerType[2].JobTableRight[0].SetForceTarget := 0;
   aRecipe[5].RecipeLayerType[1].JobTableRight[0].SetForceTarget := 0;
   aRecipe[5].RecipeLayerType[2].JobTableRight[0].SetForceTarget := 0;
   aRecipe[6].RecipeLayerType[1].JobTableRight[0].SetForceTarget := 0;
   aRecipe[6].RecipeLayerType[1].JobTableRight[1].SetForceTarget := 120;
   aRecipe[6].RecipeLayerType[2].JobTableRight[0].SetForceTarget := 0;
   aRecipe[6].RecipeLayerType[2].JobTableRight[1].SetForceTarget := 120;
   aRecipe[7].RecipeLayerType[1].JobTableRight[0].SetForceTarget := 0;
   aRecipe[7].RecipeLayerType[2].JobTableRight[0].SetForceTarget := 0;
   aRecipe[8].RecipeLayerType[1].JobTableRight[0].SetForceTarget := 0;
   aRecipe[8].RecipeLayerType[2].JobTableRight[0].SetForceTarget := 0;
   aRecipe[9].RecipeLayerType[1].JobTableRight[0].SetForceTarget := 0;
   aRecipe[9].RecipeLayerType[2].JobTableRight[0].SetForceTarget := 0;
   aRecipe[10].RecipeLayerType[1].JobTableRight[0].SetForceTarget := 0;
   aRecipe[10].RecipeLayerType[2].JobTableRight[0].SetForceTarget := 0;
   aRecipe[11].RecipeLayerType[1].JobTableRight[0].SetForceTarget := 0;
   aRecipe[11].RecipeLayerType[2].JobTableRight[0].SetForceTarget := 0;
   aRecipe[12].RecipeLayerType[1].JobTableRight[0].SetForceTarget := 0;
   aRecipe[12].RecipeLayerType[2].JobTableRight[0].SetForceTarget := 0;
   aRecipe[13].RecipeLayerType[1].JobTableRight[0].SetForceTarget := 0;
   aRecipe[13].RecipeLayerType[2].JobTableRight[0].SetForceTarget := 0;
   aRecipe[14].RecipeLayerType[1].JobTableRight[0].SetForceTarget := 0;
   aRecipe[14].RecipeLayerType[2].JobTableRight[0].SetForceTarget := 0;
   aRecipe[15].RecipeLayerType[1].JobTableRight[0].SetForceTarget := 0;
   aRecipe[15].RecipeLayerType[2].JobTableRight[0].SetForceTarget := 0;
   aRecipe[16].RecipeLayerType[1].JobTableRight[0].SetForceTarget := 0;
   aRecipe[16].RecipeLayerType[2].JobTableRight[0].SetForceTarget := 0;
   aRecipe[17].RecipeLayerType[1].JobTableRight[0].SetForceTarget := 0;
   aRecipe[17].RecipeLayerType[1].JobTableRight[1].SetForceTarget := 120;
   aRecipe[17].RecipeLayerType[2].JobTableRight[0].SetForceTarget := 0;
   aRecipe[18].RecipeLayerType[1].JobTableRight[0].SetForceTarget := 0;
   aRecipe[18].RecipeLayerType[2].JobTableRight[0].SetForceTarget := 0;
   aRecipe[19].RecipeLayerType[1].JobTableRight[0].SetForceTarget := 0;
   aRecipe[19].RecipeLayerType[2].JobTableRight[0].SetForceTarget := 0;
   aRecipe[20].RecipeLayerType[1].JobTableRight[0].SetForceTarget := 0;
   aRecipe[20].RecipeLayerType[2].JobTableRight[0].SetForceTarget := 0;
   aRecipe[21].RecipeLayerType[1].JobTableRight[0].SetForceTarget := 0;
   aRecipe[21].RecipeLayerType[2].JobTableRight[0].SetForceTarget := 0;
   aRecipe[22].RecipeLayerType[1].JobTableRight[0].SetForceTarget := 0;
   aRecipe[22].RecipeLayerType[2].JobTableRight[0].SetForceTarget := 0;
   aRecipe[23].RecipeLayerType[1].JobTableRight[0].SetForceTarget := 0;
   aRecipe[23].RecipeLayerType[2].JobTableRight[0].SetForceTarget := 0;
   aRecipe[1].RecipeLayerType[1].JobTableRight[0].SetTimeRamp := 0;
   aRecipe[1].RecipeLayerType[2].JobTableRight[0].SetTimeRamp := 0;
   aRecipe[2].RecipeLayerType[1].JobTableRight[0].SetTimeRamp := 0;
   aRecipe[2].RecipeLayerType[2].JobTableRight[0].SetTimeRamp := 0;
   aRecipe[3].RecipeLayerType[1].JobTableRight[0].SetTimeRamp := 0;
   aRecipe[3].RecipeLayerType[2].JobTableRight[0].SetTimeRamp := 0;
   aRecipe[4].RecipeLayerType[1].JobTableRight[0].SetTimeRamp := 0;
   aRecipe[4].RecipeLayerType[2].JobTableRight[0].SetTimeRamp := 0;
   aRecipe[5].RecipeLayerType[1].JobTableRight[0].SetTimeRamp := 0;
   aRecipe[5].RecipeLayerType[2].JobTableRight[0].SetTimeRamp := 0;
   aRecipe[6].RecipeLayerType[1].JobTableRight[0].SetTimeRamp := 0;
   aRecipe[6].RecipeLayerType[2].JobTableRight[0].SetTimeRamp := 0;
   aRecipe[7].RecipeLayerType[1].JobTableRight[0].SetTimeRamp := 0;
   aRecipe[7].RecipeLayerType[2].JobTableRight[0].SetTimeRamp := 0;
   aRecipe[8].RecipeLayerType[1].JobTableRight[0].SetTimeRamp := 0;
   aRecipe[8].RecipeLayerType[2].JobTableRight[0].SetTimeRamp := 0;
   aRecipe[9].RecipeLayerType[1].JobTableRight[0].SetTimeRamp := 0;
   aRecipe[9].RecipeLayerType[2].JobTableRight[0].SetTimeRamp := 0;
   aRecipe[10].RecipeLayerType[1].JobTableRight[0].SetTimeRamp := 0;
   aRecipe[10].RecipeLayerType[2].JobTableRight[0].SetTimeRamp := 0;
   aRecipe[11].RecipeLayerType[1].JobTableRight[0].SetTimeRamp := 0;
   aRecipe[11].RecipeLayerType[2].JobTableRight[0].SetTimeRamp := 0;
   aRecipe[12].RecipeLayerType[1].JobTableRight[0].SetTimeRamp := 0;
   aRecipe[12].RecipeLayerType[2].JobTableRight[0].SetTimeRamp := 0;
   aRecipe[13].RecipeLayerType[1].JobTableRight[0].SetTimeRamp := 0;
   aRecipe[13].RecipeLayerType[2].JobTableRight[0].SetTimeRamp := 0;
   aRecipe[14].RecipeLayerType[1].JobTableRight[0].SetTimeRamp := 0;
   aRecipe[14].RecipeLayerType[2].JobTableRight[0].SetTimeRamp := 0;
   aRecipe[15].RecipeLayerType[1].JobTableRight[0].SetTimeRamp := 0;
   aRecipe[15].RecipeLayerType[2].JobTableRight[0].SetTimeRamp := 0;
   aRecipe[16].RecipeLayerType[1].JobTableRight[0].SetTimeRamp := 0;
   aRecipe[16].RecipeLayerType[2].JobTableRight[0].SetTimeRamp := 0;
   aRecipe[17].RecipeLayerType[1].JobTableRight[0].SetTimeRamp := 0;
   aRecipe[17].RecipeLayerType[1].JobTableRight[1].SetTimeRamp := 2;
   aRecipe[17].RecipeLayerType[2].JobTableRight[0].SetTimeRamp := 0;
   aRecipe[18].RecipeLayerType[1].JobTableRight[0].SetTimeRamp := 0;
   aRecipe[18].RecipeLayerType[2].JobTableRight[0].SetTimeRamp := 0;
   aRecipe[19].RecipeLayerType[1].JobTableRight[0].SetTimeRamp := 0;
   aRecipe[19].RecipeLayerType[2].JobTableRight[0].SetTimeRamp := 0;
   aRecipe[20].RecipeLayerType[1].JobTableRight[0].SetTimeRamp := 0;
   aRecipe[20].RecipeLayerType[2].JobTableRight[0].SetTimeRamp := 0;
   aRecipe[21].RecipeLayerType[1].JobTableRight[0].SetTimeRamp := 0;
   aRecipe[21].RecipeLayerType[2].JobTableRight[0].SetTimeRamp := 0;
   aRecipe[22].RecipeLayerType[1].JobTableRight[0].SetTimeRamp := 0;
   aRecipe[22].RecipeLayerType[2].JobTableRight[0].SetTimeRamp := 0;
   aRecipe[23].RecipeLayerType[1].JobTableRight[0].SetTimeRamp := 0;
   aRecipe[23].RecipeLayerType[2].JobTableRight[0].SetTimeRamp := 0;
   aRecipe[1].RecipeLayerType[1].JobTableRight[0].SetSpeed := 0;
   aRecipe[1].RecipeLayerType[2].JobTableRight[0].SetSpeed := 0;
   aRecipe[2].RecipeLayerType[1].JobTableRight[0].SetSpeed := 0;
   aRecipe[2].RecipeLayerType[2].JobTableRight[0].SetSpeed := 0;
   aRecipe[3].RecipeLayerType[1].JobTableRight[0].SetSpeed := 0;
   aRecipe[3].RecipeLayerType[2].JobTableRight[0].SetSpeed := 0;
   aRecipe[4].RecipeLayerType[1].JobTableRight[0].SetSpeed := 0;
   aRecipe[4].RecipeLayerType[2].JobTableRight[0].SetSpeed := 0;
   aRecipe[5].RecipeLayerType[1].JobTableRight[0].SetSpeed := 0;
   aRecipe[5].RecipeLayerType[2].JobTableRight[0].SetSpeed := 0;
   aRecipe[6].RecipeLayerType[1].JobTableRight[0].SetSpeed := 0;
   aRecipe[6].RecipeLayerType[2].JobTableRight[0].SetSpeed := 0;
   aRecipe[7].RecipeLayerType[1].JobTableRight[0].SetSpeed := 0;
   aRecipe[7].RecipeLayerType[2].JobTableRight[0].SetSpeed := 0;
   aRecipe[8].RecipeLayerType[1].JobTableRight[0].SetSpeed := 0;
   aRecipe[8].RecipeLayerType[2].JobTableRight[0].SetSpeed := 0;
   aRecipe[9].RecipeLayerType[1].JobTableRight[0].SetSpeed := 0;
   aRecipe[9].RecipeLayerType[2].JobTableRight[0].SetSpeed := 0;
   aRecipe[10].RecipeLayerType[1].JobTableRight[0].SetSpeed := 0;
   aRecipe[10].RecipeLayerType[2].JobTableRight[0].SetSpeed := 0;
   aRecipe[11].RecipeLayerType[1].JobTableRight[0].SetSpeed := 0;
   aRecipe[11].RecipeLayerType[2].JobTableRight[0].SetSpeed := 0;
   aRecipe[12].RecipeLayerType[1].JobTableRight[0].SetSpeed := 0;
   aRecipe[12].RecipeLayerType[2].JobTableRight[0].SetSpeed := 0;
   aRecipe[13].RecipeLayerType[1].JobTableRight[0].SetSpeed := 0;
   aRecipe[13].RecipeLayerType[2].JobTableRight[0].SetSpeed := 0;
   aRecipe[14].RecipeLayerType[1].JobTableRight[0].SetSpeed := 0;
   aRecipe[14].RecipeLayerType[2].JobTableRight[0].SetSpeed := 0;
   aRecipe[15].RecipeLayerType[1].JobTableRight[0].SetSpeed := 0;
   aRecipe[15].RecipeLayerType[2].JobTableRight[0].SetSpeed := 0;
   aRecipe[16].RecipeLayerType[1].JobTableRight[0].SetSpeed := 0;
   aRecipe[16].RecipeLayerType[2].JobTableRight[0].SetSpeed := 0;
   aRecipe[17].RecipeLayerType[1].JobTableRight[0].SetSpeed := 0;
   aRecipe[17].RecipeLayerType[1].JobTableRight[1].SetSpeed := 4000;
   aRecipe[17].RecipeLayerType[2].JobTableRight[0].SetSpeed := 0;
   aRecipe[18].RecipeLayerType[1].JobTableRight[0].SetSpeed := 0;
   aRecipe[18].RecipeLayerType[2].JobTableRight[0].SetSpeed := 0;
   aRecipe[19].RecipeLayerType[1].JobTableRight[0].SetSpeed := 0;
   aRecipe[19].RecipeLayerType[2].JobTableRight[0].SetSpeed := 0;
   aRecipe[20].RecipeLayerType[1].JobTableRight[0].SetSpeed := 0;
   aRecipe[20].RecipeLayerType[2].JobTableRight[0].SetSpeed := 0;
   aRecipe[21].RecipeLayerType[1].JobTableRight[0].SetSpeed := 0;
   aRecipe[21].RecipeLayerType[2].JobTableRight[0].SetSpeed := 0;
   aRecipe[22].RecipeLayerType[1].JobTableRight[0].SetSpeed := 0;
   aRecipe[22].RecipeLayerType[2].JobTableRight[0].SetSpeed := 0;
   aRecipe[23].RecipeLayerType[1].JobTableRight[0].SetSpeed := 0;
   aRecipe[23].RecipeLayerType[2].JobTableRight[0].SetSpeed := 0;
   aRecipe[1].RecipeLayerType[1].JobTableRight[0].SetRobotSpeed := 0;
   aRecipe[1].RecipeLayerType[2].JobTableRight[0].SetRobotSpeed := 0;
   aRecipe[2].RecipeLayerType[1].JobTableRight[0].SetRobotSpeed := 0;
   aRecipe[2].RecipeLayerType[1].JobTableRight[1..2].SetRobotSpeed := 300;
   aRecipe[2].RecipeLayerType[2].JobTableRight[0].SetRobotSpeed := 0;
   aRecipe[2].RecipeLayerType[2].JobTableRight[1..2].SetRobotSpeed := 300;
   aRecipe[3].RecipeLayerType[1].JobTableRight[0].SetRobotSpeed := 0;
   aRecipe[3].RecipeLayerType[1].JobTableRight[1].SetRobotSpeed := 200;
   aRecipe[3].RecipeLayerType[1].JobTableRight[2].SetRobotSpeed := 300;
   aRecipe[3].RecipeLayerType[2].JobTableRight[0].SetRobotSpeed := 0;
   aRecipe[3].RecipeLayerType[2].JobTableRight[1].SetRobotSpeed := 300;
   aRecipe[4].RecipeLayerType[1].JobTableRight[0].SetRobotSpeed := 0;
   aRecipe[4].RecipeLayerType[2].JobTableRight[0].SetRobotSpeed := 0;
   aRecipe[5].RecipeLayerType[1].JobTableRight[0].SetRobotSpeed := 0;
   aRecipe[5].RecipeLayerType[2].JobTableRight[0].SetRobotSpeed := 0;
   aRecipe[6].RecipeLayerType[1].JobTableRight[0].SetRobotSpeed := 0;
   aRecipe[6].RecipeLayerType[2].JobTableRight[0].SetRobotSpeed := 0;
   aRecipe[7].RecipeLayerType[1].JobTableRight[0].SetRobotSpeed := 0;
   aRecipe[7].RecipeLayerType[2].JobTableRight[0].SetRobotSpeed := 0;
   aRecipe[8].RecipeLayerType[1].JobTableRight[0].SetRobotSpeed := 0;
   aRecipe[8].RecipeLayerType[2].JobTableRight[0].SetRobotSpeed := 0;
   aRecipe[9].RecipeLayerType[1].JobTableRight[0].SetRobotSpeed := 0;
   aRecipe[9].RecipeLayerType[2].JobTableRight[0].SetRobotSpeed := 0;
   aRecipe[10].RecipeLayerType[1].JobTableRight[0].SetRobotSpeed := 0;
   aRecipe[10].RecipeLayerType[2].JobTableRight[0].SetRobotSpeed := 0;
   aRecipe[11].RecipeLayerType[1].JobTableRight[0].SetRobotSpeed := 0;
   aRecipe[11].RecipeLayerType[2].JobTableRight[0].SetRobotSpeed := 0;
   aRecipe[12].RecipeLayerType[1].JobTableRight[0].SetRobotSpeed := 0;
   aRecipe[12].RecipeLayerType[2].JobTableRight[0].SetRobotSpeed := 0;
   aRecipe[13].RecipeLayerType[1].JobTableRight[0].SetRobotSpeed := 0;
   aRecipe[13].RecipeLayerType[2].JobTableRight[0].SetRobotSpeed := 0;
   aRecipe[14].RecipeLayerType[1].JobTableRight[0].SetRobotSpeed := 0;
   aRecipe[14].RecipeLayerType[2].JobTableRight[0].SetRobotSpeed := 0;
   aRecipe[15].RecipeLayerType[1].JobTableRight[0].SetRobotSpeed := 0;
   aRecipe[15].RecipeLayerType[2].JobTableRight[0].SetRobotSpeed := 0;
   aRecipe[16].RecipeLayerType[1].JobTableRight[0].SetRobotSpeed := 0;
   aRecipe[16].RecipeLayerType[2].JobTableRight[0].SetRobotSpeed := 0;
   aRecipe[17].RecipeLayerType[1].JobTableRight[0].SetRobotSpeed := 0;
   aRecipe[17].RecipeLayerType[1].JobTableRight[1].SetRobotSpeed := 150;
   aRecipe[17].RecipeLayerType[2].JobTableRight[0].SetRobotSpeed := 0;
   aRecipe[18].RecipeLayerType[1].JobTableRight[0].SetRobotSpeed := 0;
   aRecipe[18].RecipeLayerType[2].JobTableRight[0].SetRobotSpeed := 0;
   aRecipe[19].RecipeLayerType[1].JobTableRight[0].SetRobotSpeed := 0;
   aRecipe[19].RecipeLayerType[2].JobTableRight[0].SetRobotSpeed := 0;
   aRecipe[20].RecipeLayerType[1].JobTableRight[0].SetRobotSpeed := 0;
   aRecipe[20].RecipeLayerType[2].JobTableRight[0].SetRobotSpeed := 0;
   aRecipe[21].RecipeLayerType[1].JobTableRight[0].SetRobotSpeed := 0;
   aRecipe[21].RecipeLayerType[2].JobTableRight[0].SetRobotSpeed := 0;
   aRecipe[22].RecipeLayerType[1].JobTableRight[0].SetRobotSpeed := 0;
   aRecipe[22].RecipeLayerType[2].JobTableRight[0].SetRobotSpeed := 0;
   aRecipe[23].RecipeLayerType[1].JobTableRight[0].SetRobotSpeed := 0;
   aRecipe[23].RecipeLayerType[2].JobTableRight[0].SetRobotSpeed := 0;
   aRecipe[1].RecipeLayerType[1].JobTableRight[0].WornPaperDistance := 0;
   aRecipe[1].RecipeLayerType[2].JobTableRight[0].WornPaperDistance := 0;
   aRecipe[2].RecipeLayerType[1].JobTableRight[0].WornPaperDistance := 0;
   aRecipe[2].RecipeLayerType[1].JobTableRight[1].WornPaperDistance := 8;
   aRecipe[2].RecipeLayerType[1].JobTableRight[2].WornPaperDistance := 30;
   aRecipe[2].RecipeLayerType[2].JobTableRight[0].WornPaperDistance := 0;
   aRecipe[2].RecipeLayerType[2].JobTableRight[1..2].WornPaperDistance := 30;
   aRecipe[3].RecipeLayerType[1].JobTableRight[0].WornPaperDistance := 0;
   aRecipe[3].RecipeLayerType[1].JobTableRight[1..2].WornPaperDistance := 30;
   aRecipe[3].RecipeLayerType[2].JobTableRight[0].WornPaperDistance := 0;
   aRecipe[3].RecipeLayerType[2].JobTableRight[1].WornPaperDistance := 30;
   aRecipe[4].RecipeLayerType[1].JobTableRight[0].WornPaperDistance := 0;
   aRecipe[4].RecipeLayerType[2].JobTableRight[0].WornPaperDistance := 0;
   aRecipe[5].RecipeLayerType[1].JobTableRight[0].WornPaperDistance := 0;
   aRecipe[5].RecipeLayerType[2].JobTableRight[0].WornPaperDistance := 0;
   aRecipe[6].RecipeLayerType[1].JobTableRight[0].WornPaperDistance := 0;
   aRecipe[6].RecipeLayerType[2].JobTableRight[0].WornPaperDistance := 0;
   aRecipe[7].RecipeLayerType[1].JobTableRight[0].WornPaperDistance := 0;
   aRecipe[7].RecipeLayerType[2].JobTableRight[0].WornPaperDistance := 0;
   aRecipe[8].RecipeLayerType[1].JobTableRight[0].WornPaperDistance := 0;
   aRecipe[8].RecipeLayerType[2].JobTableRight[0].WornPaperDistance := 0;
   aRecipe[9].RecipeLayerType[1].JobTableRight[0].WornPaperDistance := 0;
   aRecipe[9].RecipeLayerType[2].JobTableRight[0].WornPaperDistance := 0;
   aRecipe[10].RecipeLayerType[1].JobTableRight[0].WornPaperDistance := 0;
   aRecipe[10].RecipeLayerType[2].JobTableRight[0].WornPaperDistance := 0;
   aRecipe[11].RecipeLayerType[1].JobTableRight[0].WornPaperDistance := 0;
   aRecipe[11].RecipeLayerType[2].JobTableRight[0].WornPaperDistance := 0;
   aRecipe[12].RecipeLayerType[1].JobTableRight[0].WornPaperDistance := 0;
   aRecipe[12].RecipeLayerType[2].JobTableRight[0].WornPaperDistance := 0;
   aRecipe[13].RecipeLayerType[1].JobTableRight[0].WornPaperDistance := 0;
   aRecipe[13].RecipeLayerType[2].JobTableRight[0].WornPaperDistance := 0;
   aRecipe[14].RecipeLayerType[1].JobTableRight[0].WornPaperDistance := 0;
   aRecipe[14].RecipeLayerType[2].JobTableRight[0].WornPaperDistance := 0;
   aRecipe[15].RecipeLayerType[1].JobTableRight[0].WornPaperDistance := 0;
   aRecipe[15].RecipeLayerType[2].JobTableRight[0].WornPaperDistance := 0;
   aRecipe[16].RecipeLayerType[1].JobTableRight[0].WornPaperDistance := 0;
   aRecipe[16].RecipeLayerType[2].JobTableRight[0].WornPaperDistance := 0;
   aRecipe[17].RecipeLayerType[1].JobTableRight[0].WornPaperDistance := 0;
   aRecipe[17].RecipeLayerType[2].JobTableRight[0].WornPaperDistance := 0;
   aRecipe[18].RecipeLayerType[1].JobTableRight[0].WornPaperDistance := 0;
   aRecipe[18].RecipeLayerType[2].JobTableRight[0].WornPaperDistance := 0;
   aRecipe[19].RecipeLayerType[1].JobTableRight[0].WornPaperDistance := 0;
   aRecipe[19].RecipeLayerType[2].JobTableRight[0].WornPaperDistance := 0;
   aRecipe[20].RecipeLayerType[1].JobTableRight[0].WornPaperDistance := 0;
   aRecipe[20].RecipeLayerType[2].JobTableRight[0].WornPaperDistance := 0;
   aRecipe[21].RecipeLayerType[1].JobTableRight[0].WornPaperDistance := 0;
   aRecipe[21].RecipeLayerType[2].JobTableRight[0].WornPaperDistance := 0;
   aRecipe[22].RecipeLayerType[1].JobTableRight[0].WornPaperDistance := 0;
   aRecipe[22].RecipeLayerType[2].JobTableRight[0].WornPaperDistance := 0;
   aRecipe[23].RecipeLayerType[1].JobTableRight[0].WornPaperDistance := 0;
   aRecipe[23].RecipeLayerType[2].JobTableRight[0].WornPaperDistance := 0;
   aRecipe[1].RecipeLayerType[1].JobTableRight[0].Gimball := 0;
   aRecipe[1].RecipeLayerType[2].JobTableRight[0].Gimball := 0;
   aRecipe[1].RecipeLayerType[2].JobTableRight[1].Gimball := 2;
   aRecipe[2].RecipeLayerType[1].JobTableRight[0].Gimball := 0;
   aRecipe[2].RecipeLayerType[2].JobTableRight[0].Gimball := 0;
   aRecipe[3].RecipeLayerType[1].JobTableRight[0].Gimball := 0;
   aRecipe[3].RecipeLayerType[2].JobTableRight[0].Gimball := 0;
   aRecipe[3].RecipeLayerType[2].JobTableRight[1].Gimball := 1;
   aRecipe[4].RecipeLayerType[1].JobTableRight[0].Gimball := 0;
   aRecipe[4].RecipeLayerType[2].JobTableRight[0].Gimball := 0;
   aRecipe[5].RecipeLayerType[1].JobTableRight[0].Gimball := 0;
   aRecipe[5].RecipeLayerType[2].JobTableRight[0].Gimball := 0;
   aRecipe[6].RecipeLayerType[1].JobTableRight[0].Gimball := 0;
   aRecipe[6].RecipeLayerType[2].JobTableRight[0].Gimball := 0;
   aRecipe[7].RecipeLayerType[1].JobTableRight[0].Gimball := 0;
   aRecipe[7].RecipeLayerType[2].JobTableRight[0].Gimball := 0;
   aRecipe[8].RecipeLayerType[1].JobTableRight[0].Gimball := 0;
   aRecipe[8].RecipeLayerType[2].JobTableRight[0].Gimball := 0;
   aRecipe[9].RecipeLayerType[1].JobTableRight[0].Gimball := 0;
   aRecipe[9].RecipeLayerType[2].JobTableRight[0].Gimball := 0;
   aRecipe[10].RecipeLayerType[1].JobTableRight[0].Gimball := 0;
   aRecipe[10].RecipeLayerType[2].JobTableRight[0].Gimball := 0;
   aRecipe[11].RecipeLayerType[1].JobTableRight[0].Gimball := 0;
   aRecipe[11].RecipeLayerType[2].JobTableRight[0].Gimball := 0;
   aRecipe[12].RecipeLayerType[1].JobTableRight[0].Gimball := 0;
   aRecipe[12].RecipeLayerType[2].JobTableRight[0].Gimball := 0;
   aRecipe[13].RecipeLayerType[1].JobTableRight[0].Gimball := 0;
   aRecipe[13].RecipeLayerType[2].JobTableRight[0].Gimball := 0;
   aRecipe[14].RecipeLayerType[1].JobTableRight[0].Gimball := 0;
   aRecipe[14].RecipeLayerType[2].JobTableRight[0].Gimball := 0;
   aRecipe[15].RecipeLayerType[1].JobTableRight[0].Gimball := 0;
   aRecipe[15].RecipeLayerType[2].JobTableRight[0].Gimball := 0;
   aRecipe[16].RecipeLayerType[1].JobTableRight[0].Gimball := 0;
   aRecipe[16].RecipeLayerType[2].JobTableRight[0].Gimball := 0;
   aRecipe[17].RecipeLayerType[1].JobTableRight[0].Gimball := 0;
   aRecipe[17].RecipeLayerType[1].JobTableRight[1].Gimball := 1;
   aRecipe[17].RecipeLayerType[2].JobTableRight[0].Gimball := 0;
   aRecipe[18].RecipeLayerType[1].JobTableRight[0].Gimball := 0;
   aRecipe[18].RecipeLayerType[2].JobTableRight[0].Gimball := 0;
   aRecipe[19].RecipeLayerType[1].JobTableRight[0].Gimball := 0;
   aRecipe[19].RecipeLayerType[2].JobTableRight[0].Gimball := 0;
   aRecipe[20].RecipeLayerType[1].JobTableRight[0].Gimball := 0;
   aRecipe[20].RecipeLayerType[2].JobTableRight[0].Gimball := 0;
   aRecipe[21].RecipeLayerType[1].JobTableRight[0].Gimball := 0;
   aRecipe[21].RecipeLayerType[2].JobTableRight[0].Gimball := 0;
   aRecipe[22].RecipeLayerType[1].JobTableRight[0].Gimball := 0;
   aRecipe[22].RecipeLayerType[2].JobTableRight[0].Gimball := 0;
   aRecipe[23].RecipeLayerType[1].JobTableRight[0].Gimball := 0;
   aRecipe[23].RecipeLayerType[2].JobTableRight[0].Gimball := 0;
   aRecipe[1].RecipeLayerType[2].JobTableRight[1].UnlockEccentric1 := TRUE;
   aRecipe[1].RecipeLayerType[2].JobTableRight[1].UnlockEccentric2 := TRUE;
   aRecipe[1].RecipeLayerType[2].JobTableRight[1].UnlockEccentric3 := TRUE;
END_DATA_BLOCK
